KUKA KRL data list: LAB_MINIMAL.dat

&ACCESS RVP
&REL 1
DEFDAT LAB_MINIMAL PUBLIC
  DECL E6AXIS A_HOME={A1 0,A2 -90,A3 90,A4 0,A5 0,A6 0,E1 0,E2 0,E3 0,E4 0,E5 0,E6 0}
  DECL E6POS P_START={X 1900,Y -100,Z 1200,A 180,B 0,C 180,S 2,T 2,E1 0,E2 0,E3 0,E4 0,E5 0,E6 0}
  DECL E6POS P_END={X 1900,Y 100,Z 1200,A 180,B 0,C 180,S 2,T 2,E1 0,E2 0,E3 0,E4 0,E5 0,E6 0}
ENDDAT
